FUNCTION_BLOCK FB_Btn
VAR_INPUT
	xStart:BOOL;
	xStop:BOOL;
	xReset:BOOL;
	xNextPas:BOOL;
	xAru:BOOL;
END_VAR
VAR_OUTPUT
END_VAR
VAR
END_VAR

END_FUNCTION_BLOCK

(* stored: Version 1.1.0.1, ProductVersion 3.1.4020.6
   POU FB_Btn: Id {9d1b347e-0701-4dd1-a9e2-079105cb34be}, SpecialFunc None *)
